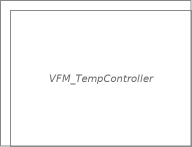
VISUALIZATION VIS_TempCtrl  // 192x147
    Frame (10,10 182x137)
        shows VFM_TempController(HMI := MAIN.Machine.TempController.HMI)
END_VISUALIZATION

(* stored: Version 1.1.0.1, ProductVersion 3.1.4024.12
   Visu VIS_TempCtrl: Id {43fbfddb-3192-4fbf-9f63-5fa566e25d72} *)
